// This function has been automatically generated from the project information.
{attribute 'signature_flag' := '1073741824'}
{attribute 'TcGenerated'}
{attribute 'no-analysis'}
FUNCTION F_GetCompany : WSTRING
VAR_INPUT
	
END_VAR

F_GetCompany := "BA";

END_FUNCTION

(* stored: Version 1.1.0.1
   POU F_GetCompany: Id {4f3d4b2a-c1d0-483a-8de2-6042ce1f0dd5}, SpecialFunc None *)
